Universal Robots PolyScope program: Put_into_box_CB3_UR5.urp

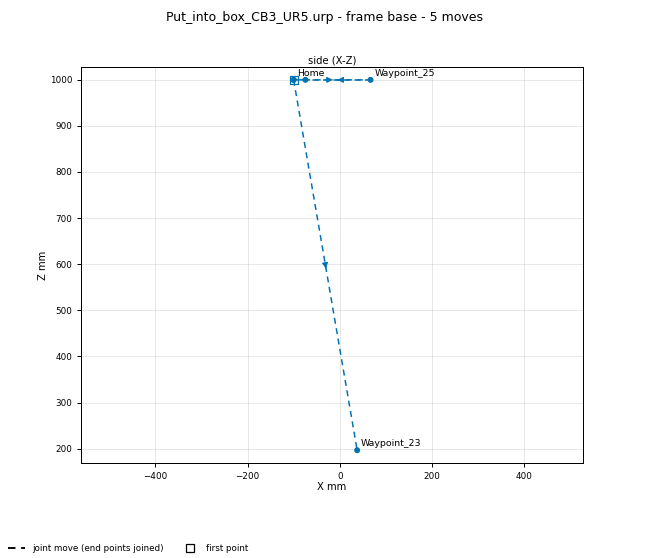
[picture p0: tool path of Put_into_box_CB3_UR5.urp in frame base, 5 of 5 moves have a stored position in this frame; points joined in program order, loops and branches not executed]
Program Put_into_box_CB3_UR5 (installation=default directory=/programs/default createdIn=3.0.0.0 lastSavedIn=3.8.0.61336 robotSerialNumber=2018359174)
Calibrated DH parameters: a=[0.000103, -0.165236, -0.391809, -0.000008, 0.000072, 0]; d=[0.08937, 126.180413, -125.613724, -0.456703, 0.094787, 0.082637]; alpha=[1.569508, -0.003108, -0.027037, 1.57048, -1.570735, 0]; deltaTheta=[0, -1.172139, 1.133037, 0.038915, 0.000034, 0.000049]
Robot Program (runOnlyOnce=true)
  Set NoAction (payload=0 tcpAsCog=true)
  MoveJ speed 10 deg/s, acceleration 80 deg/s^2 (useActiveTCP=false)
    Waypoint Home: motionParameters(blendRadius=0); TCP in base x=-99.993 y=-190.994 z=999.647 mm, rx=0.0001 ry=-2.2213 rz=2.2213 rad; joints [0, -90, 0, -90, 0, 0] deg; flange x=5.539 y=-193.713 z=1001.332 mm, rx=-0.0313 ry=2.2104 rz=-2.2041 rad
    Waypoint Waypoint_25: motionParameters(blendRadius=0); TCP in base x=66.716 y=-178.969 z=999.63 mm, rx=-0.3657 ry=2.0272 rz=-2.0272 rad; joints [20.439, -90, 0, -90, 0, 0] deg; flange x=72.838 y=-179.583 z=1001.332 mm, rx=-0.3926 ry=2.0137 rz=-2.0079 rad
    Popup Message (haltProgram=false message=Remove first bolt placed under shoulder inputType=Text)
    Waypoint Waypoint_26: motionParameters(blendRadius=0); TCP in base x=-74.498 y=-175.872 z=999.63 mm, rx=-0.4062 ry=-2.0012 rz=2.0011 rad; joints [-22.964, -90, 0, -90, 0, 0] deg; flange x=-70.478 y=-180.522 z=1001.332 mm, rx=-0.3808 ry=-2.021 rz=2.0151 rad
    Popup Message (haltProgram=false message=Remove second bolt placed under shoulder                                                                      Place protective pad between arm and base joint inputType=Text)
    Waypoint Home: motionParameters(blendRadius=0); TCP in base x=-99.993 y=-190.994 z=999.647 mm, rx=0.0001 ry=-2.2213 rz=2.2213 rad; joints [0, -90, 0, -90, 0, 0] deg; flange x=5.539 y=-193.713 z=1001.332 mm, rx=-0.0313 ry=2.2104 rz=-2.2041 rad
    Waypoint Waypoint_23: motionParameters(blendRadius=0); TCP in base x=37.68 y=-191.036 z=196.558 mm, rx=1.2057 ry=-1.2156 rz=1.2134 rad; joints [-0.055, 3.602, -163.716, -109.496, 0.049, 0.025] deg; flange x=40.767 y=-191.072 z=192.206 mm, rx=1.2307 ry=-1.2275 rz=1.2101 rad
    Popup Message (haltProgram=false message=Remove remaining bolts inputType=Text)
